{attribute 'pack_mode' := '1'}
TYPE FireIgnitor :
STRUCT
	bHeating				: BOOL;
	bBlower					: BOOL;
END_STRUCT
END_TYPE

(* stored: Version 1.1.0.1, ProductVersion 3.1.4022.18
   DUT FireIgnitor: Id {77d33174-c700-4a7e-b210-0971f25570db} *)
